FUNCTION_BLOCK ECMaster (* Service Interface Function Block Type *)
  (* Standard: 61499-2 *)
  (* Version 1.0, 2026-04-09, hyperion *)
  PACKAGE eclipse4diac::io::ethercat;
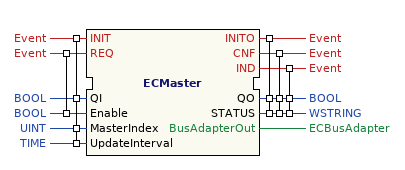
  EVENT_INPUT
    INIT WITH MasterIndex, UpdateInterval, QI; (* Service Initialization *)
    REQ WITH Enable;
  END_EVENT
  EVENT_OUTPUT
    INITO WITH QO, STATUS; (* Initialization Confirm *)
    CNF WITH QO, STATUS; (* Confirmation of Requested Service *)
    IND WITH QO, STATUS; (* Indication from Resource *)
  END_EVENT
  VAR_INPUT
    QI : BOOL;
    Enable : BOOL;
    MasterIndex : UINT;
    UpdateInterval : TIME := T#30us;
  END_VAR
  VAR_OUTPUT
    QO : BOOL; (* Event Output Qualifier *)
    STATUS : WSTRING; (* Service Status *)
  END_VAR
  PLUGS
    BusAdapterOut : eclipse4diac::io::ethercat::ECBusAdapter;
  END_PLUGS
END_FUNCTION_BLOCK
